FUNCTION_BLOCK SelectInfFeedConfig (* Basic Function Block Type *)
  (* Standard: 61499-2 *)
  (* Version 0.0, 8/24/2026, Schneider Electric, Template *)
  PACKAGE SE.Nereda;
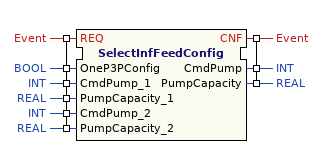
  EVENT_INPUT
    REQ WITH CmdPump_1, PumpCapacity_1, CmdPump_2, PumpCapacity_2, OneP3PConfig; (* Normal Execution Request *)
  END_EVENT
  EVENT_OUTPUT
    CNF WITH CmdPump, PumpCapacity; (* Execution Confirmation *)
  END_EVENT
  VAR_INPUT
    OneP3PConfig : BOOL; (* = FALSE : One Pump | = TRUE : 3 Pumps *)
    CmdPump_1 : INT; (* Input event qualifier *)
    PumpCapacity_1 : REAL;
    CmdPump_2 : INT;
    PumpCapacity_2 : REAL;
  END_VAR
  VAR_OUTPUT
    CmdPump : INT; (* Output event qualifier *)
    PumpCapacity : REAL;
  END_VAR
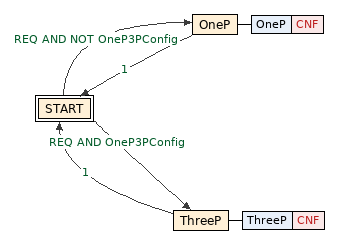
  EC_STATES
    START; (* Initial State *)
    OneP : OneP -> CNF; (* Initialization *)
    ThreeP : ThreeP -> CNF; (* Normal execution *)
  END_STATES
  EC_TRANSITIONS
    START TO OneP := REQ AND NOT OneP3PConfig;
    OneP TO START := 1;
    START TO ThreeP := REQ AND OneP3PConfig;
    ThreeP TO START := 1;
  END_TRANSITIONS
  ALGORITHM OneP IN ST: (* Initialization algorithm *)
;
CmdPump := CmdPump_1;
PumpCapacity := PumpCapacity_1;
  END_ALGORITHM
  ALGORITHM ThreeP IN ST: (* Normally executed algorithm *)
;
CmdPump := CmdPump_2;
PumpCapacity := PumpCapacity_2;
  END_ALGORITHM
END_FUNCTION_BLOCK
